% RSLogix 500 project LAB 3 SCAD BWFG_BAK118.RSS, saved by version 8.40.00.08 %
PROJECT "LAB2_BGJ"    % processor: SLC 500, 1747-L541 %

PROGRAM FILES
  LAD 2   7 rungs

DATA FILES
  O0 OUTPUT  68 elements
  I1 INPUT  68 elements
  S2 STATUS  164 elements
  B3 BINARY  10 elements
  T4 TIMER  51 elements
  C5 COUNTER  102 elements
  R6 CONTROL  1 elements
  N7 INTEGER  6 elements
  F8 FLOAT  44 elements

LADDER 2
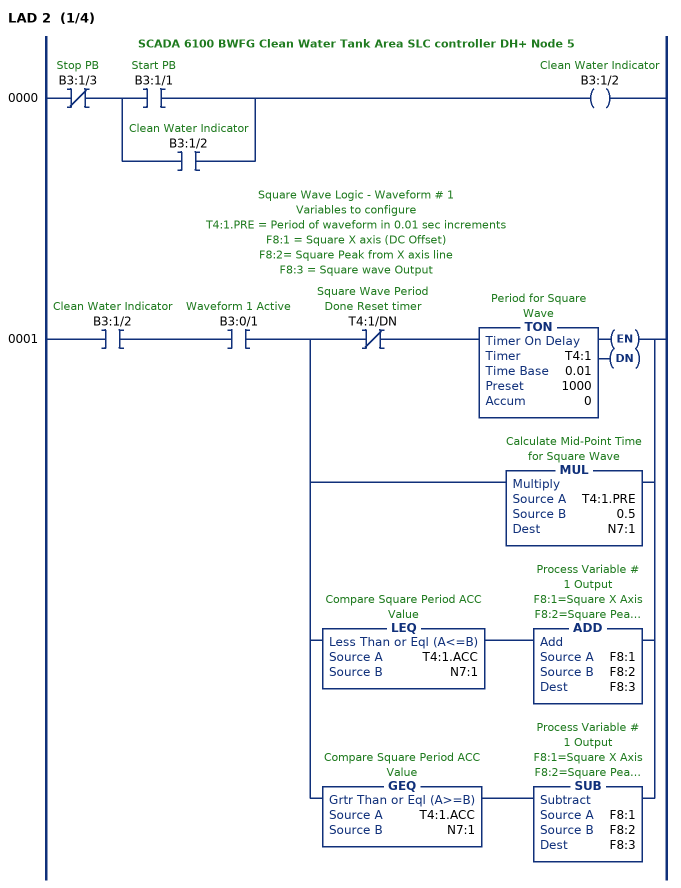
% Rung: 0 %
% TITLE: SCADA 6100 BWFG Clean Water Tank Area SLC controller DH+ Node 5 %
SOR XIO B3:1/3 BST XIC B3:1/1 NXB XIC B3:1/2 BND OTE B3:1/2 EOR
%   B3:1/3  "Stop PB" %
%   B3:1/1  "Start PB" %
%   B3:1/2  "Clean Water Indicator" %
% Rung: 1 %
% Square Wave Logic - Waveform # 1
% Variables to configure
% T4:1.PRE = Period of waveform in 0.01 sec increments
% F8:1 = Square X axis (DC Offset)
% F8:2= Square Peak from X axis line
% F8:3 = Square wave Output %
SOR XIC B3:1/2 XIC B3:0/1 BST XIO T4:1/DN TON T4:1 0.01 1000 0 NXB MUL T4:1.PRE 0.5 N7:1 NXB LEQ T4:1.ACC N7:1 ADD F8:1 F8:2 F8:3 NXB GEQ T4:1.ACC N7:1 SUB F8:1 F8:2 F8:3 BND EOR
%   B3:1/2  "Clean Water Indicator" %
%   B3:0/1  "Waveform 1 Active" %
%   T4:1/DN  "Square Wave Period Done Reset timer" %
%   T4:1  "Period for Square Wave" %
%   T4:1.PRE  "Period for Square Wave in 0.01 sec increments" %
%   N7:1  "Calculate Mid-Point Time for Square Wave" %
%   T4:1.ACC  "Compare Square Period ACC Value" %
%   F8:1  "Find Mid Point time for Square Wave" %
%   F8:2  "Square Wave Peak Parameter" %
%   F8:3  "Process Variable # 1 Output F8:1=Square X Axis F8:2=Square Peak F8:3=Waveform Output" %

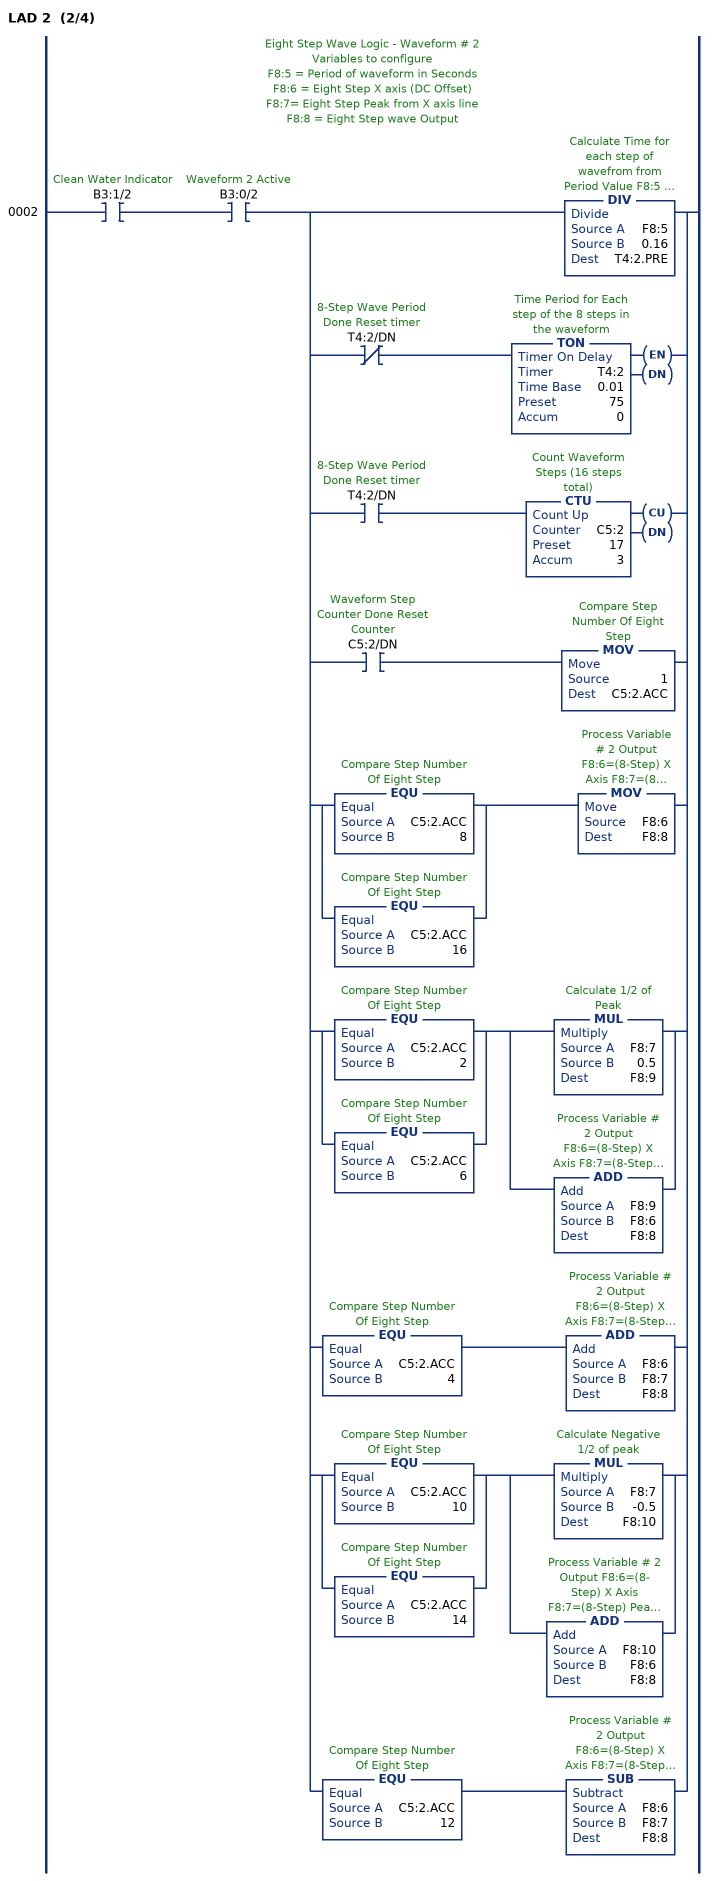
% Rung: 2 %
% Eight Step Wave Logic - Waveform # 2
% Variables to configure
% F8:5 = Period of waveform in Seconds
% F8:6 = Eight Step X axis (DC Offset)
% F8:7= Eight Step Peak from X axis line
% F8:8 = Eight Step wave Output %
SOR XIC B3:1/2 XIC B3:0/2 BST DIV F8:5 0.16 T4:2.PRE NXB XIO T4:2/DN TON T4:2 0.01 75 0 NXB XIC T4:2/DN CTU C5:2 17 3 NXB XIC C5:2/DN MOV 1 C5:2.ACC NXB BST EQU C5:2.ACC 8 NXB EQU C5:2.ACC 16 BND MOV F8:6 F8:8 NXB BST EQU C5:2.ACC 2 NXB EQU C5:2.ACC 6 BND BST MUL F8:7 0.5 F8:9 NXB ADD F8:9 F8:6 F8:8 BND NXB EQU C5:2.ACC 4 ADD F8:6 F8:7 F8:8 NXB BST EQU C5:2.ACC 10 NXB EQU C5:2.ACC 14 BND BST MUL F8:7 -0.5 F8:10 NXB ADD F8:10 F8:6 F8:8 BND NXB EQU C5:2.ACC 12 SUB F8:6 F8:7 F8:8 BND EOR
%   B3:1/2  "Clean Water Indicator" %
%   B3:0/2  "Waveform 2 Active" %
%   T4:2.PRE  "Calculate Time for each step of wavefrom from Period Value F8:5 = Period in Sec" %
%   T4:2/DN  "8-Step Wave Period Done Reset timer" %
%   T4:2  "Time Period for Each step of the 8 steps in the waveform" %
%   C5:2  "Count Waveform Steps (16 steps total)" %
%   C5:2/DN  "Waveform Step Counter Done Reset Counter" %
%   C5:2.ACC  "Compare Step Number Of Eight Step" %
%   F8:6  "X-Axis Value For Eight Step" %
%   F8:8  "Process Variable # 2 Output F8:6=(8-Step) X Axis F8:7=(8-Step) Peak F8:8=(8-Step) Output" %
%   F8:7  "Eight Step Peak" %
%   F8:9  "Calculate 1/2 of Peak" %
%   F8:10  "Calculate Negative 1/2 of peak" %

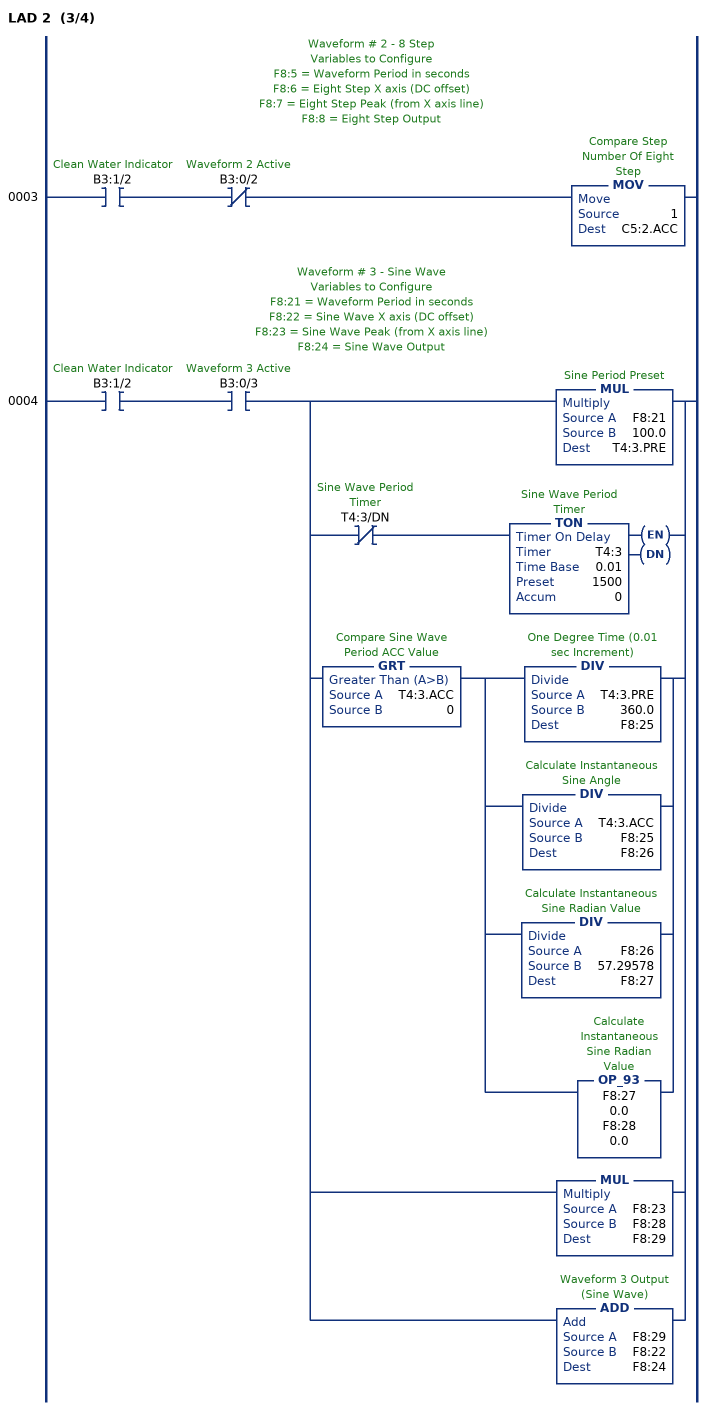
% Rung: 3 %
% Waveform # 2 - 8 Step
% Variables to Configure
% F8:5 = Waveform Period in seconds
% F8:6 = Eight Step X axis (DC offset)
% F8:7 = Eight Step Peak (from X axis line)
% F8:8 = Eight Step Output %
SOR XIC B3:1/2 XIO B3:0/2 MOV 1 C5:2.ACC EOR
%   B3:1/2  "Clean Water Indicator" %
%   B3:0/2  "Waveform 2 Active" %
%   C5:2.ACC  "Compare Step Number Of Eight Step" %
% Rung: 4 %
% Waveform # 3 - Sine Wave
% Variables to Configure
% F8:21 = Waveform Period in seconds
% F8:22 = Sine Wave X axis (DC offset)
% F8:23 = Sine Wave Peak (from X axis line)
% F8:24 = Sine Wave Output %
SOR XIC B3:1/2 XIC B3:0/3 BST MUL F8:21 100.0 T4:3.PRE NXB XIO T4:3/DN TON T4:3 0.01 1500 0 NXB GRT T4:3.ACC 0 BST DIV T4:3.PRE 360.0 F8:25 NXB DIV T4:3.ACC F8:25 F8:26 NXB DIV F8:26 57.29578 F8:27 NXB OP_93 F8:27 0.0 F8:28 0.0 BND NXB MUL F8:23 F8:28 F8:29 NXB ADD F8:29 F8:22 F8:24 BND EOR
%   B3:1/2  "Clean Water Indicator" %
%   B3:0/3  "Waveform 3 Active" %
%   T4:3.PRE  "Sine Period Preset" %
%   T4:3  "Sine Wave Period Timer" %
%   T4:3.ACC  "Compare Sine Wave Period ACC Value" %
%   F8:25  "One Degree Time (0.01 sec Increment)" %
%   F8:26  "Calculate Instantaneous Sine Angle" %
%   F8:27  "Calculate Instantaneous Sine Radian Value" %
%   F8:28  "Calculate Sine of Instantaneous Angle" %
%   F8:23  "Sine Peak Parameter" %
%   F8:22  "Sine X Axis Parameter" %
%   F8:24  "Waveform 3 Output (Sine Wave)" %

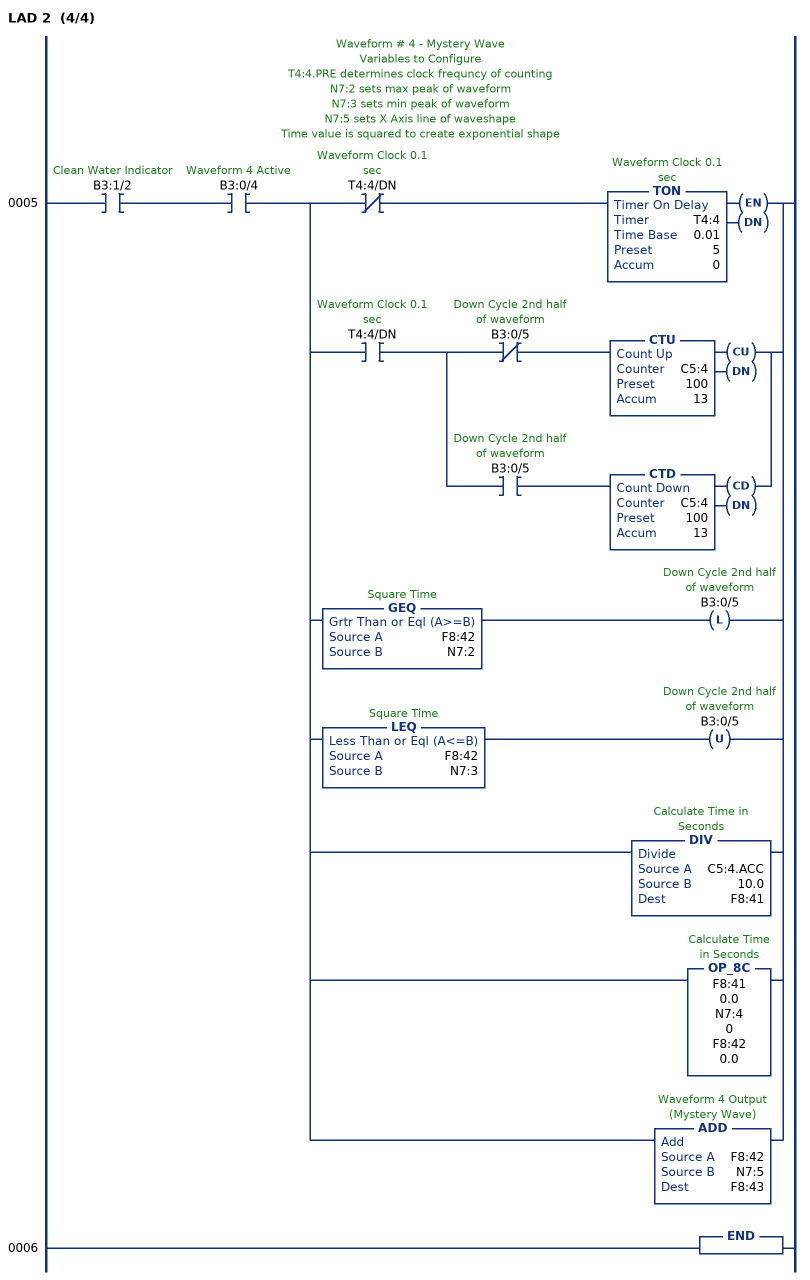
% Rung: 5 %
% Waveform # 4 - Mystery Wave
% Variables to Configure
% T4:4.PRE determines clock frequncy of counting
% N7:2 sets max peak of waveform
% N7:3 sets min peak of waveform
% N7:5 sets X Axis line of waveshape
% Time value is squared to create exponential shape %
SOR XIC B3:1/2 XIC B3:0/4 BST XIO T4:4/DN TON T4:4 0.01 5 0 NXB XIC T4:4/DN BST XIO B3:0/5 CTU C5:4 100 13 NXB XIC B3:0/5 CTD C5:4 100 13 BND NXB GEQ F8:42 N7:2 OTL B3:0/5 NXB LEQ F8:42 N7:3 OTU B3:0/5 NXB DIV C5:4.ACC 10.0 F8:41 NXB OP_8C F8:41 0.0 N7:4 0 F8:42 0.0 NXB ADD F8:42 N7:5 F8:43 BND EOR
%   B3:1/2  "Clean Water Indicator" %
%   B3:0/4  "Waveform 4 Active" %
%   T4:4  "Waveform Clock 0.1 sec" %
%   B3:0/5  "Down Cycle 2nd half of waveform" %
%   F8:42  "Square Time" %
%   F8:41  "Calculate Time in Seconds" %
%   F8:43  "Waveform 4 Output (Mystery Wave)" %
% Rung: 6 %
SOR END EOR

OTHER DOCUMENTED ADDRESSES
  B3:0/0  "HMI_OZONE_CON_PB"
  B3:0/10  "PART 1 START/STOP MEMORY"
  B3:1/4  "PART 2 START/STOP MEMORY CASCADED TIMERS"
  B3:1/14  "PART 3 START/STOP MEMORY"
  C5:1  "PART 3 UP/DOWN COUNTER"
  C5:1/CU  "COUNT UP ENABLED CTU IS ENERGIZED"
  C5:1/DN  "ACC IS GREATER THAN OR EQUAL TO PRE VALUE (25 IN THIS EXAMPLE)"
  C5:5  "PART 3 UP/DOWN COUNTER"
  C5:5.ACC  "SEND COUNTER ACCUMULATOR TO LED DISPLAY"
  C5:5.PRE  "LOAD COUNT PRESET FROM THUMBWHEEL"
  C5:10  "PART 3 UP/DOWN COUNTER"
  C5:10.ACC  "COUNTER ACC TO LED DISPLAY"
  C5:10.PRE  "LOAD COUNT PRESET FROM THUMBWHEEL"
  C5:10/CD  "CTD INSTRUCTION ENABLED"
  C5:10/CU  "CTU INSTRUCTION ENABLED"
  C5:10/DN  "COUNT ACC>=PRE (DONE)"
  C5:10/OV  "COUNTER ACC >32767 (OVERFLOW) ACC WRAPS TO ZERO"
  C5:10/UN  "COUNTER ACC LESS THAN -32768 ACC WRAPS TO ZERO"
  C5:31  "1ST COUNTER HORN ON TIME COUNTS 0.3 SEC (6 X 0.05 SEC)"
  C5:31/DN  "1ST COUNTER DONE ENGAGE 2ND COUNTER"
  C5:32  "2ND COUNTER HORN OFF TIME COUNTS 0.6 SEC (12 X 0.05 SEC)"
  C5:32/DN  "2ND COUNTER DONE RESET COUNTERS"
  C5:33  "PART 3 UP/DOWN COUNTER"
  C5:33.ACC  "DISPLAY UP/DOWN COUNTER ACC ON LED DISPLAY"
  C5:33.PRE  "LOAD UP/DOWN COUNTER PRESET FROM THUMBWHEEL"
  C5:33/DN  "UP/DOWN COUNTER DONE ENGAGE HORN"
  C5:34  "HORN CYCLE COUNTER STOP HORN AFTER 5 CYCLES"
  C5:100  "MINUTES FOR 24 HR CLOCK"
  C5:100.ACC  "DISPLAY MINUTES ON LED DISPLAY"
  C5:100/DN  "INDEX HOUR COUNTER EVERY 60 MINUTES"
  C5:101  "HOURS FOR 24 HR CLOCK"
  C5:101/DN  "RESET HOUR COUNT AT BEGINNING OF A NEW DAY"
  I:1.0/0  "1PBLT-BUTTON RESET COUNTER"
  I:1.0/1  "2PBLT BUTTON PART1: LOAD TIMER PART2: LOAD RED TIME PART3: LOAD HORN ON TIME"
  I:1.0/2  "3PBLT BUTTON PART 2: LOAD GREEN TIME PART 3: LOAD HORN OFF TIME"
  I:1.0/3  "4PBLT BUTTON PART 2: LOAD AMBER TIME PART3: LOAD COUNTER PRESET"
  I:1.0/4  "5PB START BUTTON"
  I:1.0/5  "6PB COUNT UP"
  I:1.0/6  "7PB STOP BUTTON"
  I:1.0/7  "8PB STOP BUTTON"
  I:1.0/8  "COUNT UP PB"
  I:1.0/9  "COUNT DOWN PB"
  I:1.0/10  "3SS POS 1 POSITION"
  I:1.0/11  "3SS POS 3 POSITION"
  I:1.0/12  "SET MINUTES FROM THUMBWHELL WHEN PRESSED"
  I:1.0/13  "SET HOURS FROM THUMBWHEEL WHEN PRESSED"
  I:1.0/14  "SHOW SECONDS ON LED DISPLAY"
  I:1.0/15  "SHOW MINUTES ON LED DISPLAY"
  I:3.0  "LOAD ACCUMULATOR FROM THUMBWHEEL"
  I:5.0/0  "SHOW HOURS ON LED DISPLAY"
  O:2.0/0  "GREEN LIGHT"
  O:2.0/1  "AMBER LIGHT"
  O:2.0/2  "RED LIGHT"
  O:2.0/3  "FLASHING LIGHT"
  O:2.0/4  "1LT GREEN LIGHT"
  O:2.0/5  "2LT FLASHING LIGHT"
  O:2.0/6  "3LT RED LIGHT FLASH ON/OFF"
  O:2.0/7  "4LT GREEN STACK LIGHT"
  O:2.0/8  "5LT AMBER STACK LIGHT"
  O:2.0/9  "6LT RED STACK LIGHT"
  O:2.0/10  "1AH HORN"
  O:2.0/11  "COUNTER UNDERFLOW"
  O:4.0  "ACCUMULATOR TO LED DISPLAY"
  T4:1.ACC/6  "0.64 SEC FLASHING BIT OF FREE RUN TIMER"
  T4:2/TT  "O.75 SEC FLASHER WHILE STAGE 1 IS TIMING"
  T4:5  "AMBER LIGHT TIMER"
  T4:5/DN  "AMBER TIME DONE START RED"
  T4:6  "RED LIGHT TIMER"
  T4:6/DN  "RED TIME DONE RESET FOR NEXT CYCLE"
  T4:10  "PART 1 FREE RUN TIMER"
  T4:10.ACC  "PART 1 FREE RUN TIMER TO LED DISPLAY"
  T4:10.PRE  "LOAD FREE RUN TIMER FROM THUMBWHEEL"
  T4:10/DN  "FREE RUN TIMER DONE RESET FOR NEXT CYCLE"
  T4:11  "PART 1 FREE RUNNING TIMER"
  T4:11.ACC  "DISPLAY TIMER ACC ON LED DISPLAY"
  T4:11.ACC/5  "0.32 SEC FLASHER"
  T4:11.ACC/6  "0.32 SEC FLASHER"
  T4:11.PRE  "LOAD FREE RUN TIMER PREST FROM THUMBWHEEL"
  T4:11/DN  "TIMER DONE RESET"
  T4:12  "PART 2 GREEN LIGHT CASCADE TIMER 2"
  T4:12.PRE  "LOAD GREEN TIME PRESET FROM THUMBWHEEL"
  T4:12/DN  "GREEN LIGHT TIMER DONE"
  T4:12/TT  "GREEN LIGHT TIMER TIMING"
  T4:13  "PART 2 AMBER LIGHT CASCADE TIMER 3"
  T4:13.PRE  "LOAD AMBER TIME PRESET FROM THUMBWHEEL"
  T4:13/DN  "LAST CASCADE TIMER DONE RESET CYCLE"
  T4:13/TT  "AMBER LIGHT TIMER TIMING"
  T4:20  "PART 3 HORN TIMER 2.25 SEC"
  T4:20/DN  "HORN TIME DONE"
  T4:21  "PART 2 RED LIGHT TIME CASCADED TIMER 1"
  T4:21.PRE  "LOAD RED TIME PRESET FROM THUMBWHEEL"
  T4:21/DN  "RED TIME DONE START GREEN TIMER"
  T4:21/TT  "ENERGIZE RED LIGHT"
  T4:22  "PART 2 GREEN LIGHT CASCADE TIMER 2"
  T4:22.PRE  "LOAD GREEN TIME PRESET FROM THUMBWHEEL"
  T4:22/DN  "GREEN TIME DONE START AMBER TIMER"
  T4:22/TT  "ENERGIZE GREEN LIGHT"
  T4:23  "PART 2 AMBER LIGHT CASCADE TIMER 3"
  T4:23.PRE  "LOAD AMBER TIME PRESET FROM THUMBWHEEL"
  T4:23/DN  "LAST CASCADE TIMER DONE RESET CYCLE"
  T4:23/TT  "ENERGIZE AMBER LIGHT"
  T4:24  "LIGHT ON TIME"
  T4:24/DN  "1ST CASCADE TIME DONE START 2ND TIMER"
  T4:24/TT  "LIGHT ON TIME"
  T4:25  "LIGHT OFF TIME"
  T4:25/DN  "2ND CASCADE TIMER DONE RESET CIRCUIT"
  T4:30  "PART 3 HORN TIMER 2.75 SEC"
  T4:30/DN  "HORN TIME DONE SHUT OFF HORN"
  T4:31  "0.05 SEC FREE RUN TIMER"
  T4:31/DN  "TIME DONE RESET FREE RUN TIMER AND INDEX COUNTER"
  T4:32  "HORN ON TIME"
  T4:32.PRE  "LOAD HORN ON TIME FROM THUMBWHEEL"
  T4:32/DN  "HORN ON TIME DONE"
  T4:33  "HORN OFF TIME"
  T4:33.PRE  "LOAD HORN OFF TIME FROM THUBWHEEL"
  T4:33/DN  "HORN OFF TIME DONE RESET TIMERS"
  T4:50  "SECONDS FOR 24 HR CLOCK"
  T4:50/DN  "RESET FREE RUN TIMER"

OTHER INSTRUCTION COMMENTS
  C5:1 RES  "PART 3 RESET COUNTER TO ZERO"
  C5:10 RES  "PART 3 RESET COUNTER TO ZERO"
  T4:50/DN XIC  "INDEX MINUTE COUNTER EVERY 60 SECONDS"
  C5:100 RES  "RESET MINUTE COUNT EVERY HOUR"
  C5:101 RES  "RESET HOUR COUNT START OF NEW DAY"
  C5:100.ACC FRD  "MINUTES FOR 24 HR CLOCK"

COMMENTS NOT ATTACHED TO A CURRENT RUNG
  B3:1/14: PART 3 - HORN TIMER AND UP/DOWN COUNTER, THUMBWHEEL AND LED DISPLAY
  B3:1/4: PART 2 - CASCADED TIMERS AND SIMPLE TRAFFIC LIGHT
  B3:0/10: PART 1 - FREE RUN TIMER PLUS THUMBWHEEL AND LED DISPLAY / Lab Solution - Brent Brooks - Winter 2008
  B3:0/0: PAGE TITLE TO START INTERNAL MEMORY BIT ON A NEW PAGE WHEN PRINTING / INTERNAL MEMORY BIT B3/0 FROM FILE B3 - RUNG COMMENT
  T4:1: FREE RUNNING TIMER CIRCUIT
  O:2.0/3: FLASHING LIGHT FROM ACC BIT OF FREE RUNNING TIMER
  T4:2: CASCADED TIMER CIRCUIT CONSISTING OF TWO TIMING STAGES WITH T4:2 AND T4:3
  B3:0/2: PART 2 - CASCADED TIMERS AND TRAFFIC LIGHT
  B3:0/3: PART 3 - HORN TIMER AND UP/DOWN COUNTER AND THUMBWHEEL AND LED DISPLAY

DATA TABLE (non-zero values as saved)
DATA B3
% B3:0 % 0X0000 0X4000 0X0000 0X0000 0X0000 0X0000 0X0000 0X0000 0X0000 0X0000
DATA T4
% .PRE .ACC %
% T4:1 % 1000 0
% T4:2 % 75 0
% T4:3 % 1500 0
% T4:4 % 5 0
% T4:5 % 5 0
% T4:6 % 20 0
% T4:10 % 1500 0
% T4:11 % 128 0
% T4:12 % 500 0
% T4:13 % 200 0
% T4:20 % 225 0
% T4:21 % 525 0
% T4:22 % 245 0
% T4:23 % 175 0
% T4:24 % 75 0
% T4:25 % 50 0
% T4:30 % 275 0
% T4:31 % 5 0
% T4:32 % 25 25
% T4:33 % 150 30
% T4:50 % 60 0
DATA C5
% .PRE .ACC %
% C5:1 % 25 0
% C5:2 % 17 3
% C5:4 % 100 13
% C5:5 % 25 0
% C5:10 % 25 0
% C5:31 % 6 1
% C5:32 % 12 0
% C5:33 % 10 10
% C5:34 % 6 6
% C5:100 % 60 35
% C5:101 % 24 10
